// TIA Portal V16 export
// export: Created 2021-10-20T17:21:35.7534833Z, ExportSetting WithDefaults, DisplayName Totally Integrated Automation Portal, DisplayVersion V16, DisplayName TIA Portal Version Control Interface, DisplayVersion V16, DisplayName TIA Portal Openness, DisplayVersion V16, DisplayName TIA Portal Teamcenter Gateway, DisplayVersion V16, DisplayName SINAMICS Startdrive Advanced, DisplayVersion V16, DisplayName SINAMICS Startdrive G130, G150, S120, S150, SINAMICS MV, S210, DisplayVersion V16, DisplayName SINAMICS Startdrive G110M, G120, G120C, G120D, G120P, DisplayVersion V16, DisplayName STEP 7 Professional, DisplayVersion V16, DisplayName STEP 7 Safety, DisplayVersion V16, DisplayName WinCC Advanced, DisplayVersion V16
FUNCTION_BLOCK "Mapped Bits"   // FB6, LAD
TITLE = Mapped Bits for HMI
{ S7_Optimized_Access := 'TRUE' }
VERSION : 0.1
// stored: AutoNumber true, IsIECCheckEnabled false, IsRetainMemResEnabled false, MemoryReserve 100, SetENOAutomatically false, UDAEnableTagReadback false
BEGIN

REGION Network 1: Venting HMI bits
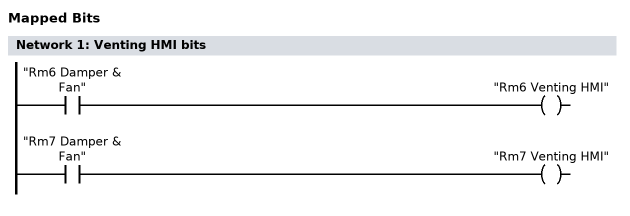
   RUNG wire#powerrail
      Contact( "Rm6 Damper & Fan" )
      Coil( "Rm6 Venting HMI" )
   END_RUNG
   RUNG wire#powerrail
      Contact( "Rm7 Damper & Fan" )
      Coil( "Rm7 Venting HMI" )
   END_RUNG
   // the same network as SCL:
   "Rm6 Venting HMI" := "Rm6 Damper & Fan";
   "Rm7 Venting HMI" := "Rm7 Damper & Fan";
END_REGION
END_FUNCTION_BLOCK
